# EPICS substitutions: iocBoot/iocTomoScan_13BM_MCS/tomoScan.substitutions
file "$(TOP)/db/tomoScan.template"
{
pattern
{  P,      R,    CAMERA,    FILE_PLUGIN,   ROTATION,  SAMPLE_X,  SAMPLE_Y,      CLOSE_SHUTTER,        CLOSE_VALUE,        OPEN_SHUTTER,         OPEN_VALUE}
{13BMDPG2:, TS:, 13BMDPG2:, 13BMDPG2:HDF1:, 13BMD:m38, 13BMD:m85, 13BMD:m90, 13BMA:CloseBMDShutter.PROC,    1,        13BMA:OpenBMDShutter.PROC,      1}
}

file "$(TOP)/db/tomoScan_13BM_MCS.template"
{
pattern
{  P,      R,      MCS}
{13BMDPG2:, TS: 13BMD:MCS1:}
}

file "$(TOP)/db/tomoScan_13BM.template"
{
pattern
{  P,      R,       BEAM_READY,      READY_VALUE,}
{13BMDPG2:, TS:, 13BMA:mono_pid1Locked,     1,}
}
